FUNCTION_BLOCK FB_Pump
VAR_INPUT
	bStartCmd	: BOOL;
	bStopCmd	: BOOL;
END_VAR
VAR_OUTPUT
END_VAR
VAR
	_bIsOn		: BOOL;
	_rFlowRate	: REAL;
END_VAR

PROPERTY bError : BOOL
GET
//ERROR STATE IF 'bStartCmd' IS ON AND PUMP IS NOT ON
bError	:= bStartCmd AND NOT bIsOn;
END_GET
SET
END_SET
END_PROPERTY

PROPERTY bIsOn : BOOL
GET
bIsOn	:= _bIsOn;
END_GET
SET
_bIsOn	:= bIsOn;
END_SET
END_PROPERTY

METHOD Execute : BOOL
VAR_INPUT
END_VAR
//CHECK ON STATE
IF bStartCmd THEN
	bIsOn		:= TRUE;
ELSIF bStopCmd THEN
	bIsOn		:= FALSE;
END_IF
END_METHOD

METHOD FB_init : BOOL
VAR_INPUT
	bInitRetains : BOOL; // if TRUE, the retain variables are initialized (warm start / cold start)
	bInCopyCode : BOOL;  // if TRUE, the instance afterwards gets moved into the copy code (online change)
END_VAR
//FLOW RATE NITIALIZATION
rFlowRate	:= 50.0;
END_METHOD

PROPERTY rFlowRate : REAL
GET
rFlowRate	:= _rFlowRate;
END_GET
SET
_rFlowRate	:= rFlowRate;
END_SET
END_PROPERTY

METHOD SetFlowRate : BOOL
VAR_INPUT
	rRate	: REAL;
END_VAR
//SET RATE
rFlowRate	:= rRate;
END_METHOD

ACTION Stop:
//SET COMMANDS TO STOP
bStartCmd	:= FALSE;
bStopCmd	:= TRUE;
END_ACTION

END_FUNCTION_BLOCK

(* stored: Version 1.1.0.1, ProductVersion 3.1.4024.12
   POU FB_Pump: Id {b98365dc-24f0-47c3-9e64-858b2355d9b2}, SpecialFunc None
   Property bError: Id {c756b756-88ce-408d-aa93-ded232701c24}
   Get Get: Id {600f7e5c-89b6-4434-b45a-59ac25a65c11}
   Set Set: Id {c58e52ff-cf32-4305-bb4a-b01c86457804}
   Property bIsOn: Id {ea638808-ea05-4482-b1c7-c3f710b620fe}
   Get Get: Id {9c3d3d13-6a5e-4a2e-881b-d839e8aec501}
   Set Set: Id {b158cd58-19c9-4679-84e8-8a82477d3962}
   Method Execute: Id {1d4f8a3a-cfbb-42c7-876e-a93d9f256b72}
   Method FB_init: Id {6e55d4e2-b785-4b6d-8e8f-440e6e5bae7a}
   Property rFlowRate: Id {2c9952d7-7cf3-4e54-9da4-22409be8e6a2}
   Get Get: Id {3d432222-aa82-48b2-aeb6-7b00981993c3}
   Set Set: Id {dc5f821f-2ec7-4ae6-aec8-26503b318fe9}
   Method SetFlowRate: Id {111e02f2-6038-4a6c-9c9d-60237c808e50}
   Action Stop: Id {04c11640-edd6-4d96-8d47-bee47abe1576} *)
